FUNCTION_BLOCK APPEND_STRING_2 (* Service Interface Function Block Type *)
  (* Description: Copyright (c) 2012 Profactor GmbH This program and the accompanying materials are made available under the terms of the Eclipse Public License 2.0 which is available at https://www.eclipse.org/legal/epl-2.0/ SPDX-License-Identifier: EPL-2.0 *)
  (* Version 1.0, 2012-09-05, Matthias Plasch, Profactor GmbH *)
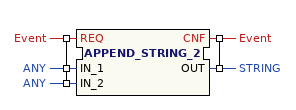
  EVENT_INPUT
    REQ WITH IN_1, IN_2; (* Service Request *)
  END_EVENT
  EVENT_OUTPUT
    CNF WITH OUT; (* Confirmation of Requested Service *)
  END_EVENT
  VAR_INPUT
    IN_1 : ANY; (* Data Input 1 (value is converted to String) *)
    IN_2 : ANY; (* Data Input 2 (value is converted to String) *)
  END_VAR
  VAR_OUTPUT
    OUT : STRING; (* Concatenated output string *)
  END_VAR
END_FUNCTION_BLOCK
